// TIA Portal V16 export
// export: Created 2022-08-05T18:22:19.1297051Z, ExportSetting WithDefaults, DisplayName Totally Integrated Automation Portal, DisplayVersion V16, DisplayName TIA Portal Version Control Interface, DisplayVersion V16, DisplayName TIA Portal Openness, DisplayVersion V16, DisplayName SINAMICS Startdrive Advanced, DisplayVersion V16, DisplayName SINAMICS Startdrive G130, G150, S120, S150, SINAMICS MV, S210, DisplayVersion V16, DisplayName SINAMICS Startdrive G110M, G120, G120C, G120D, G120P, DisplayVersion V16, DisplayName STEP 7 Professional, DisplayVersion V16, DisplayName STEP 7 Safety, DisplayVersion V16, DisplayName WinCC Professional, DisplayVersion V16
ORGANIZATION_BLOCK "TwoWay_Switch(XOR)"   // OB1, LAD, ProgramCycle
TITLE = "Main Program Sweep (Cycle)"
{ S7_Optimized_Access := 'TRUE' }
VERSION : 0.1
// stored: AutoNumber true, IsIECCheckEnabled false, SetENOAutomatically false
   VAR_INPUT
      Initial_Call : Bool;   // Initial call of this OB
      Remanence : Bool;   // =True, if remanent data are available
   END_VAR
BEGIN

REGION Network 1
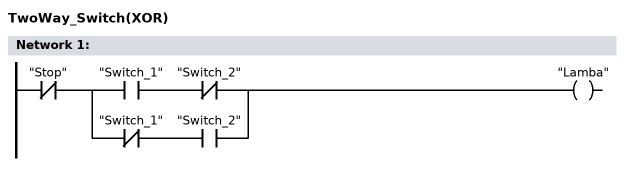
   RUNG wire#powerrail
      I_Contact( "Stop" )
      wire#w1
      Contact( "Switch_1" )
      I_Contact( "Switch_2" )
      wire#w2
      Coil( "Lamba" )
   END_RUNG
   RUNG wire#w1
      I_Contact( "Switch_1" )
      Contact( "Switch_2" )
   END_RUNG wire#w2
   // the same network as SCL:
   "Lamba" := NOT "Stop" AND (("Switch_1" AND NOT "Switch_2") OR (NOT "Switch_1" AND "Switch_2"));
END_REGION
END_ORGANIZATION_BLOCK
